TYPE ST_UPSGET :
STRUCT
	r_InputVoltage		:	REAL;
	r_OutputVoltage		:	REAL;
	r_BatteryVoltage	:	REAL;
	ui_SOC				:	UINT;
	
	b_ChargerActive		:	BOOL;
	b_SystemOnBattery	:	BOOL;
	
	UPSPowerDemand	:  	ST_PowerDemand;
	
	Events			:	ST_UPSEvents;
END_STRUCT
END_TYPE

(* stored: Version 1.1.0.1, ProductVersion 3.1.4024.12
   DUT ST_UPSGET: Id {797933e8-58da-45ca-b216-51b4073f8130} *)
